TYPE PositionValues :
STRUCT
	q1			:LREAL;
	q2			:LREAL;
	q3			:LREAL;
	q4			:LREAL;
	q5			:LREAL;
	q6			:LREAL;
END_STRUCT
END_TYPE

(* stored: Version 1.1.0.1
   DUT PositionValues: Id {20a04407-5b99-4bbd-9f81-469b44942134} *)
